        ToWin32ErrorCode := Win32ErrorCodes.ERROR_DS_DRA_INCONSISTENT_DIT;
    8444:
        ToWin32ErrorCode := Win32ErrorCodes.ERROR_DS_DRA_CONNECTION_FAILED;
    8445:
        ToWin32ErrorCode := Win32ErrorCodes.ERROR_DS_DRA_BAD_INSTANCE_TYPE;
    8446:
        ToWin32ErrorCode := Win32ErrorCodes.ERROR_DS_DRA_OUT_OF_MEM;
    8447:
        ToWin32ErrorCode := Win32ErrorCodes.ERROR_DS_DRA_MAIL_PROBLEM;
    8448:
        ToWin32ErrorCode := Win32ErrorCodes.ERROR_DS_DRA_REF_ALREADY_EXISTS;
    8449:
        ToWin32ErrorCode := Win32ErrorCodes.ERROR_DS_DRA_REF_NOT_FOUND;
    8450:
        ToWin32ErrorCode := Win32ErrorCodes.ERROR_DS_DRA_OBJ_IS_REP_SOURCE;
    8451:
        ToWin32ErrorCode := Win32ErrorCodes.ERROR_DS_DRA_DB_ERROR;
    8452:
        ToWin32ErrorCode := Win32ErrorCodes.ERROR_DS_DRA_NO_REPLICA;
    8453:
        ToWin32ErrorCode := Win32ErrorCodes.ERROR_DS_DRA_ACCESS_DENIED;
    8454:
        ToWin32ErrorCode := Win32ErrorCodes.ERROR_DS_DRA_NOT_SUPPORTED;
    8455:
        ToWin32ErrorCode := Win32ErrorCodes.ERROR_DS_DRA_RPC_CANCELLED;
    8456:
        ToWin32ErrorCode := Win32ErrorCodes.ERROR_DS_DRA_SOURCE_DISABLED;
    8457:
        ToWin32ErrorCode := Win32ErrorCodes.ERROR_DS_DRA_SINK_DISABLED;
    8458:
        ToWin32ErrorCode := Win32ErrorCodes.ERROR_DS_DRA_NAME_COLLISION;
    8459:
        ToWin32ErrorCode := Win32ErrorCodes.ERROR_DS_DRA_SOURCE_REINSTALLED;
    8460:
        ToWin32ErrorCode := Win32ErrorCodes.ERROR_DS_DRA_MISSING_PARENT;
    8461:
        ToWin32ErrorCode := Win32ErrorCodes.ERROR_DS_DRA_PREEMPTED;
    8462:
        ToWin32ErrorCode := Win32ErrorCodes.ERROR_DS_DRA_ABANDON_SYNC;
    8463:
        ToWin32ErrorCode := Win32ErrorCodes.ERROR_DS_DRA_SHUTDOWN;
    8464:
        ToWin32ErrorCode := Win32ErrorCodes.ERROR_DS_DRA_INCOMPATIBLE_PARTIAL_SET;
    8465:
        ToWin32ErrorCode := Win32ErrorCodes.ERROR_DS_DRA_SOURCE_IS_PARTIAL_REPLICA;
    8466:
        ToWin32ErrorCode := Win32ErrorCodes.ERROR_DS_DRA_EXTN_CONNECTION_FAILED;
    8467:
        ToWin32ErrorCode := Win32ErrorCodes.ERROR_DS_INSTALL_SCHEMA_MISMATCH;
    8468:
        ToWin32ErrorCode := Win32ErrorCodes.ERROR_DS_DUP_LINK_ID;
    8469:
        ToWin32ErrorCode := Win32ErrorCodes.ERROR_DS_NAME_ERROR_RESOLVING;
    8470:
        ToWin32ErrorCode := Win32ErrorCodes.ERROR_DS_NAME_ERROR_NOT_FOUND;
    8471:
        ToWin32ErrorCode := Win32ErrorCodes.ERROR_DS_NAME_ERROR_NOT_UNIQUE;
    8472:
        ToWin32ErrorCode := Win32ErrorCodes.ERROR_DS_NAME_ERROR_NO_MAPPING;
    8473:
        ToWin32ErrorCode := Win32ErrorCodes.ERROR_DS_NAME_ERROR_DOMAIN_ONLY;
    8474:
        ToWin32ErrorCode := Win32ErrorCodes.ERROR_DS_NAME_ERROR_NO_SYNTACTICAL_MAPPING;
    8475:
        ToWin32ErrorCode := Win32ErrorCodes.ERROR_DS_CONSTRUCTED_ATT_MOD;
    8476:
        ToWin32ErrorCode := Win32ErrorCodes.ERROR_DS_WRONG_OM_OBJ_CLASS;
    8477:
        ToWin32ErrorCode := Win32ErrorCodes.ERROR_DS_DRA_REPL_PENDING;
    8478:
        ToWin32ErrorCode := Win32ErrorCodes.ERROR_DS_DS_REQUIRED;
    8479:
        ToWin32ErrorCode := Win32ErrorCodes.ERROR_DS_INVALID_LDAP_DISPLAY_NAME;
    8480:
        ToWin32ErrorCode := Win32ErrorCodes.ERROR_DS_NON_BASE_SEARCH;
    8481:
        ToWin32ErrorCode := Win32ErrorCodes.ERROR_DS_CANT_RETRIEVE_ATTS;
    8482:
        ToWin32ErrorCode := Win32ErrorCodes.ERROR_DS_BACKLINK_WITHOUT_LINK;
    8483:
        ToWin32ErrorCode := Win32ErrorCodes.ERROR_DS_EPOCH_MISMATCH;
    8484:
        ToWin32ErrorCode := Win32ErrorCodes.ERROR_DS_SRC_NAME_MISMATCH;
    8485:
        ToWin32ErrorCode := Win32ErrorCodes.ERROR_DS_SRC_AND_DST_NC_IDENTICAL;
    8486:
        ToWin32ErrorCode := Win32ErrorCodes.ERROR_DS_DST_NC_MISMATCH;
    8487:
        ToWin32ErrorCode := Win32ErrorCodes.ERROR_DS_NOT_AUTHORITIVE_FOR_DST_NC;
    8488:
        ToWin32ErrorCode := Win32ErrorCodes.ERROR_DS_SRC_GUID_MISMATCH;
    8489:
        ToWin32ErrorCode := Win32ErrorCodes.ERROR_DS_CANT_MOVE_DELETED_OBJECT;
    8490:
        ToWin32ErrorCode := Win32ErrorCodes.ERROR_DS_PDC_OPERATION_IN_PROGRESS;
    8491:
        ToWin32ErrorCode := Win32ErrorCodes.ERROR_DS_CROSS_DOMAIN_CLEANUP_REQD;
    8492:
        ToWin32ErrorCode := Win32ErrorCodes.ERROR_DS_ILLEGAL_XDOM_MOVE_OPERATION;
    8493:
        ToWin32ErrorCode := Win32ErrorCodes.ERROR_DS_CANT_WITH_ACCT_GROUP_MEMBERSHPS;
    8494:
        ToWin32ErrorCode := Win32ErrorCodes.ERROR_DS_NC_MUST_HAVE_NC_PARENT;
    8495:
        ToWin32ErrorCode := Win32ErrorCodes.ERROR_DS_CR_IMPOSSIBLE_TO_VALIDATE;
    8496:
        ToWin32ErrorCode := Win32ErrorCodes.ERROR_DS_DST_DOMAIN_NOT_NATIVE;
    8497:
        ToWin32ErrorCode := Win32ErrorCodes.ERROR_DS_MISSING_INFRASTRUCTURE_CONTAINER;
    8498:
        ToWin32ErrorCode := Win32ErrorCodes.ERROR_DS_CANT_MOVE_ACCOUNT_GROUP;
    8499:
        ToWin32ErrorCode := Win32ErrorCodes.ERROR_DS_CANT_MOVE_RESOURCE_GROUP;
    8500:
        ToWin32ErrorCode := Win32ErrorCodes.ERROR_DS_INVALID_SEARCH_FLAG;
    8501:
        ToWin32ErrorCode := Win32ErrorCodes.ERROR_DS_NO_TREE_DELETE_ABOVE_NC;
    8502:
        ToWin32ErrorCode := Win32ErrorCodes.ERROR_DS_COULDNT_LOCK_TREE_FOR_DELETE;
    8503:
        ToWin32ErrorCode := Win32ErrorCodes.ERROR_DS_COULDNT_IDENTIFY_OBJECTS_FOR_TREE_DELETE;
    8504:
        ToWin32ErrorCode := Win32ErrorCodes.ERROR_DS_SAM_INIT_FAILURE;
    8505:
        ToWin32ErrorCode := Win32ErrorCodes.ERROR_DS_SENSITIVE_GROUP_VIOLATION;
    8506:
        ToWin32ErrorCode := Win32ErrorCodes.ERROR_DS_CANT_MOD_PRIMARYGROUPID;
    8507:
        ToWin32ErrorCode := Win32ErrorCodes.ERROR_DS_ILLEGAL_BASE_SCHEMA_MOD;
    8508:
        ToWin32ErrorCode := Win32ErrorCodes.ERROR_DS_NONSAFE_SCHEMA_CHANGE;
    8509:
        ToWin32ErrorCode := Win32ErrorCodes.ERROR_DS_SCHEMA_UPDATE_DISALLOWED;
    8510:
        ToWin32ErrorCode := Win32ErrorCodes.ERROR_DS_CANT_CREATE_UNDER_SCHEMA;
    8511:
        ToWin32ErrorCode := Win32ErrorCodes.ERROR_DS_INSTALL_NO_SRC_SCH_VERSION;
    8512:
        ToWin32ErrorCode := Win32ErrorCodes.ERROR_DS_INSTALL_NO_SCH_VERSION_IN_INIFILE;
    8513:
        ToWin32ErrorCode := Win32ErrorCodes.ERROR_DS_INVALID_GROUP_TYPE;
    8514:
        ToWin32ErrorCode := Win32ErrorCodes.ERROR_DS_NO_NEST_GLOBALGROUP_IN_MIXEDDOMAIN;
    8515:
        ToWin32ErrorCode := Win32ErrorCodes.ERROR_DS_NO_NEST_LOCALGROUP_IN_MIXEDDOMAIN;
    8516:
        ToWin32ErrorCode := Win32ErrorCodes.ERROR_DS_GLOBAL_CANT_HAVE_LOCAL_MEMBER;
    8517:
        ToWin32ErrorCode := Win32ErrorCodes.ERROR_DS_GLOBAL_CANT_HAVE_UNIVERSAL_MEMBER;
    8518:
        ToWin32ErrorCode := Win32ErrorCodes.ERROR_DS_UNIVERSAL_CANT_HAVE_LOCAL_MEMBER;
    8519:
        ToWin32ErrorCode := Win32ErrorCodes.ERROR_DS_GLOBAL_CANT_HAVE_CROSSDOMAIN_MEMBER;
    8520:
        ToWin32ErrorCode := Win32ErrorCodes.ERROR_DS_LOCAL_CANT_HAVE_CROSSDOMAIN_LOCAL_MEMBER;
    8521:
        ToWin32ErrorCode := Win32ErrorCodes.ERROR_DS_HAVE_PRIMARY_MEMBERS;
    8522:
        ToWin32ErrorCode := Win32ErrorCodes.ERROR_DS_STRING_SD_CONVERSION_FAILED;
    8523:
        ToWin32ErrorCode := Win32ErrorCodes.ERROR_DS_NAMING_MASTER_GC;
    8524:
        ToWin32ErrorCode := Win32ErrorCodes.ERROR_DS_LOOKUP_FAILURE;
    8525:
        ToWin32ErrorCode := Win32ErrorCodes.ERROR_DS_COULDNT_UPDATE_SPNS;
    8526:
        ToWin32ErrorCode := Win32ErrorCodes.ERROR_DS_CANT_RETRIEVE_SD;
    8527:
        ToWin32ErrorCode := Win32ErrorCodes.ERROR_DS_KEY_NOT_UNIQUE;
    8528:
        ToWin32ErrorCode := Win32ErrorCodes.ERROR_DS_WRONG_LINKED_ATT_SYNTAX;
    8529:
        ToWin32ErrorCode := Win32ErrorCodes.ERROR_DS_SAM_NEED_BOOTKEY_PASSWORD;
    8530:
        ToWin32ErrorCode := Win32ErrorCodes.ERROR_DS_SAM_NEED_BOOTKEY_FLOPPY;
    8531:
        ToWin32ErrorCode := Win32ErrorCodes.ERROR_DS_CANT_START;
    8532:
        ToWin32ErrorCode := Win32ErrorCodes.ERROR_DS_INIT_FAILURE;
    8533:
        ToWin32ErrorCode := Win32ErrorCodes.ERROR_DS_NO_PKT_PRIVACY_ON_CONNECTION;
    8534:
        ToWin32ErrorCode := Win32ErrorCodes.ERROR_DS_SOURCE_DOMAIN_IN_FOREST;
    8535:
        ToWin32ErrorCode := Win32ErrorCodes.ERROR_DS_DESTINATION_DOMAIN_NOT_IN_FOREST;
    8536:
        ToWin32ErrorCode := Win32ErrorCodes.ERROR_DS_DESTINATION_AUDITING_NOT_ENABLED;
    8537:
        ToWin32ErrorCode := Win32ErrorCodes.ERROR_DS_CANT_FIND_DC_FOR_SRC_DOMAIN;
    8538:
        ToWin32ErrorCode := Win32ErrorCodes.ERROR_DS_SRC_OBJ_NOT_GROUP_OR_USER;
    8539:
        ToWin32ErrorCode := Win32ErrorCodes.ERROR_DS_SRC_SID_EXISTS_IN_FOREST;
    8540:
        ToWin32ErrorCode := Win32ErrorCodes.ERROR_DS_SRC_AND_DST_OBJECT_CLASS_MISMATCH;
    8541:
        ToWin32ErrorCode := Win32ErrorCodes.ERROR_SAM_INIT_FAILURE;
    8542:
        ToWin32ErrorCode := Win32ErrorCodes.ERROR_DS_DRA_SCHEMA_INFO_SHIP;
    8543:
        ToWin32ErrorCode := Win32ErrorCodes.ERROR_DS_DRA_SCHEMA_CONFLICT;
    8544:
        ToWin32ErrorCode := Win32ErrorCodes.ERROR_DS_DRA_EARLIER_SCHEMA_CONLICT;
    8545:
        ToWin32ErrorCode := Win32ErrorCodes.ERROR_DS_DRA_OBJ_NC_MISMATCH;
    8546:
        ToWin32ErrorCode := Win32ErrorCodes.ERROR_DS_NC_STILL_HAS_DSAS;
    8547:
        ToWin32ErrorCode := Win32ErrorCodes.ERROR_DS_GC_REQUIRED;
    8548:
        ToWin32ErrorCode := Win32ErrorCodes.ERROR_DS_LOCAL_MEMBER_OF_LOCAL_ONLY;
    8549:
        ToWin32ErrorCode := Win32ErrorCodes.ERROR_DS_NO_FPO_IN_UNIVERSAL_GROUPS;
    8550:
        ToWin32ErrorCode := Win32ErrorCodes.ERROR_DS_CANT_ADD_TO_GC;
    8551:
        ToWin32ErrorCode := Win32ErrorCodes.ERROR_DS_NO_CHECKPOINT_WITH_PDC;
    8552:
        ToWin32ErrorCode := Win32ErrorCodes.ERROR_DS_SOURCE_AUDITING_NOT_ENABLED;
    8553:
        ToWin32ErrorCode := Win32ErrorCodes.ERROR_DS_CANT_CREATE_IN_NONDOMAIN_NC;
    8554:
        ToWin32ErrorCode := Win32ErrorCodes.ERROR_DS_INVALID_NAME_FOR_SPN;
    8555:
        ToWin32ErrorCode := Win32ErrorCodes.ERROR_DS_FILTER_USES_CONTRUCTED_ATTRS;
    8556:
        ToWin32ErrorCode := Win32ErrorCodes.ERROR_DS_UNICODEPWD_NOT_IN_QUOTES;
    8557:
        ToWin32ErrorCode := Win32ErrorCodes.ERROR_DS_MACHINE_ACCOUNT_QUOTA_EXCEEDED;
    8558:
        ToWin32ErrorCode := Win32ErrorCodes.ERROR_DS_MUST_BE_RUN_ON_DST_DC;
    8559:
        ToWin32ErrorCode := Win32ErrorCodes.ERROR_DS_SRC_DC_MUST_BE_SP4_OR_GREATER;
    8560:
        ToWin32ErrorCode := Win32ErrorCodes.ERROR_DS_CANT_TREE_DELETE_CRITICAL_OBJ;
    8561:
        ToWin32ErrorCode := Win32ErrorCodes.ERROR_DS_INIT_FAILURE_CONSOLE;
    8562:
        ToWin32ErrorCode := Win32ErrorCodes.ERROR_DS_SAM_INIT_FAILURE_CONSOLE;
    8563:
        ToWin32ErrorCode := Win32ErrorCodes.ERROR_DS_FOREST_VERSION_TOO_HIGH;
    8564:
        ToWin32ErrorCode := Win32ErrorCodes.ERROR_DS_DOMAIN_VERSION_TOO_HIGH;
    8565:
        ToWin32ErrorCode := Win32ErrorCodes.ERROR_DS_FOREST_VERSION_TOO_LOW;
    8566:
        ToWin32ErrorCode := Win32ErrorCodes.ERROR_DS_DOMAIN_VERSION_TOO_LOW;
    8567:
        ToWin32ErrorCode := Win32ErrorCodes.ERROR_DS_INCOMPATIBLE_VERSION;
    8568:
        ToWin32ErrorCode := Win32ErrorCodes.ERROR_DS_LOW_DSA_VERSION;
    8569:
        ToWin32ErrorCode := Win32ErrorCodes.ERROR_DS_NO_BEHAVIOR_VERSION_IN_MIXEDDOMAIN;
    8570:
        ToWin32ErrorCode := Win32ErrorCodes.ERROR_DS_NOT_SUPPORTED_SORT_ORDER;
    8571:
        ToWin32ErrorCode := Win32ErrorCodes.ERROR_DS_NAME_NOT_UNIQUE;
    8572:
        ToWin32ErrorCode := Win32ErrorCodes.ERROR_DS_MACHINE_ACCOUNT_CREATED_PRENT4;
    8573:
        ToWin32ErrorCode := Win32ErrorCodes.ERROR_DS_OUT_OF_VERSION_STORE;
    8574:
        ToWin32ErrorCode := Win32ErrorCodes.ERROR_DS_INCOMPATIBLE_CONTROLS_USED;
    8575:
        ToWin32ErrorCode := Win32ErrorCodes.ERROR_DS_NO_REF_DOMAIN;
    8576:
        ToWin32ErrorCode := Win32ErrorCodes.ERROR_DS_RESERVED_LINK_ID;
    8577:
        ToWin32ErrorCode := Win32ErrorCodes.ERROR_DS_LINK_ID_NOT_AVAILABLE;
    8578:
        ToWin32ErrorCode := Win32ErrorCodes.ERROR_DS_AG_CANT_HAVE_UNIVERSAL_MEMBER;
    8579:
        ToWin32ErrorCode := Win32ErrorCodes.ERROR_DS_MODIFYDN_DISALLOWED_BY_INSTANCE_TYPE;
    8580:
        ToWin32ErrorCode := Win32ErrorCodes.ERROR_DS_NO_OBJECT_MOVE_IN_SCHEMA_NC;
    8581:
        ToWin32ErrorCode := Win32ErrorCodes.ERROR_DS_MODIFYDN_DISALLOWED_BY_FLAG;
    8582:
        ToWin32ErrorCode := Win32ErrorCodes.ERROR_DS_MODIFYDN_WRONG_GRANDPARENT;
    8583:
        ToWin32ErrorCode := Win32ErrorCodes.ERROR_DS_NAME_ERROR_TRUST_REFERRAL;
    8584:
        ToWin32ErrorCode := Win32ErrorCodes.ERROR_NOT_SUPPORTED_ON_STANDARD_SERVER;
    8585:
        ToWin32ErrorCode := Win32ErrorCodes.ERROR_DS_CANT_ACCESS_REMOTE_PART_OF_AD;
    8586:
        ToWin32ErrorCode := Win32ErrorCodes.ERROR_DS_CR_IMPOSSIBLE_TO_VALIDATE_V2;
    8587:
        ToWin32ErrorCode := Win32ErrorCodes.ERROR_DS_THREAD_LIMIT_EXCEEDED;
    8588:
        ToWin32ErrorCode := Win32ErrorCodes.ERROR_DS_NOT_CLOSEST;
    9001:
        ToWin32ErrorCode := Win32ErrorCodes.DNS_ERROR_RCODE_FORMAT_ERROR;
    9002:
        ToWin32ErrorCode := Win32ErrorCodes.DNS_ERROR_RCODE_SERVER_FAILURE;
    9003:
        ToWin32ErrorCode := Win32ErrorCodes.DNS_ERROR_RCODE_NAME_ERROR;
    9004:
        ToWin32ErrorCode := Win32ErrorCodes.DNS_ERROR_RCODE_NOT_IMPLEMENTED;
    9005:
        ToWin32ErrorCode := Win32ErrorCodes.DNS_ERROR_RCODE_REFUSED;
    9006:
        ToWin32ErrorCode := Win32ErrorCodes.DNS_ERROR_RCODE_YXDOMAIN;
    9007:
        ToWin32ErrorCode := Win32ErrorCodes.DNS_ERROR_RCODE_YXRRSET;
    9008:
        ToWin32ErrorCode := Win32ErrorCodes.DNS_ERROR_RCODE_NXRRSET;
    9009:
        ToWin32ErrorCode := Win32ErrorCodes.DNS_ERROR_RCODE_NOTAUTH;
    9010:
        ToWin32ErrorCode := Win32ErrorCodes.DNS_ERROR_RCODE_NOTZONE;
    9016:
        ToWin32ErrorCode := Win32ErrorCodes.DNS_ERROR_RCODE_BADSIG;
    9017:
        ToWin32ErrorCode := Win32ErrorCodes.DNS_ERROR_RCODE_BADKEY;
    9018:
        ToWin32ErrorCode := Win32ErrorCodes.DNS_ERROR_RCODE_BADTIME;
    9501:
        ToWin32ErrorCode := Win32ErrorCodes.DNS_INFO_NO_RECORDS;
    9502:
        ToWin32ErrorCode := Win32ErrorCodes.DNS_ERROR_BAD_PACKET;
    9503:
        ToWin32ErrorCode := Win32ErrorCodes.DNS_ERROR_NO_PACKET;
    9504:
        ToWin32ErrorCode := Win32ErrorCodes.DNS_ERROR_RCODE;
    9505:
        ToWin32ErrorCode := Win32ErrorCodes.DNS_ERROR_UNSECURE_PACKET;
    9551:
        ToWin32ErrorCode := Win32ErrorCodes.DNS_ERROR_INVALID_TYPE;
    9552:
        ToWin32ErrorCode := Win32ErrorCodes.DNS_ERROR_INVALID_IP_ADDRESS;
    9553:
        ToWin32ErrorCode := Win32ErrorCodes.DNS_ERROR_INVALID_PROPERTY;
    9554:
        ToWin32ErrorCode := Win32ErrorCodes.DNS_ERROR_TRY_AGAIN_LATER;
    9555:
        ToWin32ErrorCode := Win32ErrorCodes.DNS_ERROR_NOT_UNIQUE;
    9556:
        ToWin32ErrorCode := Win32ErrorCodes.DNS_ERROR_NON_RFC_NAME;
    9557:
        ToWin32ErrorCode := Win32ErrorCodes.DNS_STATUS_FQDN;
    9558:
        ToWin32ErrorCode := Win32ErrorCodes.DNS_STATUS_DOTTED_NAME;
    9559:
        ToWin32ErrorCode := Win32ErrorCodes.DNS_STATUS_SINGLE_PART_NAME;
    9560:
        ToWin32ErrorCode := Win32ErrorCodes.DNS_ERROR_INVALID_NAME_CHAR;
    9561:
        ToWin32ErrorCode := Win32ErrorCodes.DNS_ERROR_NUMERIC_NAME;
    9601:
        ToWin32ErrorCode := Win32ErrorCodes.DNS_ERROR_ZONE_DOES_NOT_EXIST;
    9602:
        ToWin32ErrorCode := Win32ErrorCodes.DNS_ERROR_NO_ZONE_INFO;
    9603:
        ToWin32ErrorCode := Win32ErrorCodes.DNS_ERROR_INVALID_ZONE_OPERATION;
    9604:
        ToWin32ErrorCode := Win32ErrorCodes.DNS_ERROR_ZONE_CONFIGURATION_ERROR;
    9605:
        ToWin32ErrorCode := Win32ErrorCodes.DNS_ERROR_ZONE_HAS_NO_SOA_RECORD;
    9606:
        ToWin32ErrorCode := Win32ErrorCodes.DNS_ERROR_ZONE_HAS_NO_NS_RECORDS;
    9607:
        ToWin32ErrorCode := Win32ErrorCodes.DNS_ERROR_ZONE_LOCKED;
    9608:
        ToWin32ErrorCode := Win32ErrorCodes.DNS_ERROR_ZONE_CREATION_FAILED;
    9609:
        ToWin32ErrorCode := Win32ErrorCodes.DNS_ERROR_ZONE_ALREADY_EXISTS;
    9610:
        ToWin32ErrorCode := Win32ErrorCodes.DNS_ERROR_AUTOZONE_ALREADY_EXISTS;
    9611:
        ToWin32ErrorCode := Win32ErrorCodes.DNS_ERROR_INVALID_ZONE_TYPE;
    9612:
        ToWin32ErrorCode := Win32ErrorCodes.DNS_ERROR_SECONDARY_REQUIRES_MASTER_IP;
    9613:
        ToWin32ErrorCode := Win32ErrorCodes.DNS_ERROR_ZONE_NOT_SECONDARY;
    9614:
        ToWin32ErrorCode := Win32ErrorCodes.DNS_ERROR_NEED_SECONDARY_ADDRESSES;
    9615:
        ToWin32ErrorCode := Win32ErrorCodes.DNS_ERROR_WINS_INIT_FAILED;
    9616:
        ToWin32ErrorCode := Win32ErrorCodes.DNS_ERROR_NEED_WINS_SERVERS;
    9617:
        ToWin32ErrorCode := Win32ErrorCodes.DNS_ERROR_NBSTAT_INIT_FAILED;
    9618:
        ToWin32ErrorCode := Win32ErrorCodes.DNS_ERROR_SOA_DELETE_INVALID;
    9619:
        ToWin32ErrorCode := Win32ErrorCodes.DNS_ERROR_FORWARDER_ALREADY_EXISTS;
    9651:
        ToWin32ErrorCode := Win32ErrorCodes.DNS_ERROR_PRIMARY_REQUIRES_DATAFILE;
    9652:
        ToWin32ErrorCode := Win32ErrorCodes.DNS_ERROR_INVALID_DATAFILE_NAME;
    9653:
        ToWin32ErrorCode := Win32ErrorCodes.DNS_ERROR_DATAFILE_OPEN_FAILURE;
    9654:
        ToWin32ErrorCode := Win32ErrorCodes.DNS_ERROR_FILE_WRITEBACK_FAILED;
    9655:
        ToWin32ErrorCode := Win32ErrorCodes.DNS_ERROR_DATAFILE_PARSING;
    9701:
        ToWin32ErrorCode := Win32ErrorCodes.DNS_ERROR_RECORD_DOES_NOT_EXIST;
    9702:
        ToWin32ErrorCode := Win32ErrorCodes.DNS_ERROR_RECORD_FORMAT;
    9703:
        ToWin32ErrorCode := Win32ErrorCodes.DNS_ERROR_NODE_CREATION_FAILED;
    9704:
        ToWin32ErrorCode := Win32ErrorCodes.DNS_ERROR_UNKNOWN_RECORD_TYPE;
    9705:
        ToWin32ErrorCode := Win32ErrorCodes.DNS_ERROR_RECORD_TIMED_OUT;
    9706:
        ToWin32ErrorCode := Win32ErrorCodes.DNS_ERROR_NAME_NOT_IN_ZONE;
    9707:
        ToWin32ErrorCode := Win32ErrorCodes.DNS_ERROR_CNAME_LOOP;
    9708:
        ToWin32ErrorCode := Win32ErrorCodes.DNS_ERROR_NODE_IS_CNAME;
    9709:
        ToWin32ErrorCode := Win32ErrorCodes.DNS_ERROR_CNAME_COLLISION;
    9710:
        ToWin32ErrorCode := Win32ErrorCodes.DNS_ERROR_RECORD_ONLY_AT_ZONE_ROOT;
    9711:
        ToWin32ErrorCode := Win32ErrorCodes.DNS_ERROR_RECORD_ALREADY_EXISTS;
    9712:
        ToWin32ErrorCode := Win32ErrorCodes.DNS_ERROR_SECONDARY_DATA;
    9713:
        ToWin32ErrorCode := Win32ErrorCodes.DNS_ERROR_NO_CREATE_CACHE_DATA;
    9714:
        ToWin32ErrorCode := Win32ErrorCodes.DNS_ERROR_NAME_DOES_NOT_EXIST;
    9715:
        ToWin32ErrorCode := Win32ErrorCodes.DNS_WARNING_PTR_CREATE_FAILED;
    9716:
        ToWin32ErrorCode := Win32ErrorCodes.DNS_WARNING_DOMAIN_UNDELETED;
    9717:
        ToWin32ErrorCode := Win32ErrorCodes.DNS_ERROR_DS_UNAVAILABLE;
    9718:
        ToWin32ErrorCode := Win32ErrorCodes.DNS_ERROR_DS_ZONE_ALREADY_EXISTS;
    9719:
        ToWin32ErrorCode := Win32ErrorCodes.DNS_ERROR_NO_BOOTFILE_IF_DS_ZONE;
    9751:
        ToWin32ErrorCode := Win32ErrorCodes.DNS_INFO_AXFR_COMPLETE;
    9752:
        ToWin32ErrorCode := Win32ErrorCodes.DNS_ERROR_AXFR;
    9753:
        ToWin32ErrorCode := Win32ErrorCodes.DNS_INFO_ADDED_LOCAL_WINS;
    9801:
        ToWin32ErrorCode := Win32ErrorCodes.DNS_STATUS_CONTINUE_NEEDED;
    9851:
        ToWin32ErrorCode := Win32ErrorCodes.DNS_ERROR_NO_TCPIP;
    9852:
        ToWin32ErrorCode := Win32ErrorCodes.DNS_ERROR_NO_DNS_SERVERS;
    9901:
        ToWin32ErrorCode := Win32ErrorCodes.DNS_ERROR_DP_DOES_NOT_EXIST;
    9902:
        ToWin32ErrorCode := Win32ErrorCodes.DNS_ERROR_DP_ALREADY_EXISTS;
    9903:
        ToWin32ErrorCode := Win32ErrorCodes.DNS_ERROR_DP_NOT_ENLISTED;
    9904:
        ToWin32ErrorCode := Win32ErrorCodes.DNS_ERROR_DP_ALREADY_ENLISTED;
    10004:
        ToWin32ErrorCode := Win32ErrorCodes.WSAEINTR;
    10009:
        ToWin32ErrorCode := Win32ErrorCodes.WSAEBADF;
    10013:
        ToWin32ErrorCode := Win32ErrorCodes.WSAEACCES;
    10014:
        ToWin32ErrorCode := Win32ErrorCodes.WSAEFAULT;
    10022:
        ToWin32ErrorCode := Win32ErrorCodes.WSAEINVAL;
    10024:
        ToWin32ErrorCode := Win32ErrorCodes.WSAEMFILE;
    10035:
        ToWin32ErrorCode := Win32ErrorCodes.WSAEWOULDBLOCK;
    10036:
        ToWin32ErrorCode := Win32ErrorCodes.WSAEINPROGRESS;
    10037:
        ToWin32ErrorCode := Win32ErrorCodes.WSAEALREADY;
    10038:
        ToWin32ErrorCode := Win32ErrorCodes.WSAENOTSOCK;
    10039:
        ToWin32ErrorCode := Win32ErrorCodes.WSAEDESTADDRREQ;
    10040:
        ToWin32ErrorCode := Win32ErrorCodes.WSAEMSGSIZE;
    10041:
        ToWin32ErrorCode := Win32ErrorCodes.WSAEPROTOTYPE;
    10042:
        ToWin32ErrorCode := Win32ErrorCodes.WSAENOPROTOOPT;
    10043:
        ToWin32ErrorCode := Win32ErrorCodes.WSAEPROTONOSUPPORT;
    10044:
        ToWin32ErrorCode := Win32ErrorCodes.WSAESOCKTNOSUPPORT;
    10045:
        ToWin32ErrorCode := Win32ErrorCodes.WSAEOPNOTSUPP;
    10046:
        ToWin32ErrorCode := Win32ErrorCodes.WSAEPFNOSUPPORT;
    10047:
        ToWin32ErrorCode := Win32ErrorCodes.WSAEAFNOSUPPORT;
    10048:
        ToWin32ErrorCode := Win32ErrorCodes.WSAEADDRINUSE;
    10049:
        ToWin32ErrorCode := Win32ErrorCodes.WSAEADDRNOTAVAIL;
    10050:
        ToWin32ErrorCode := Win32ErrorCodes.WSAENETDOWN;
    10051:
        ToWin32ErrorCode := Win32ErrorCodes.WSAENETUNREACH;
    10052:
        ToWin32ErrorCode := Win32ErrorCodes.WSAENETRESET;
    10053:
        ToWin32ErrorCode := Win32ErrorCodes.WSAECONNABORTED;
    10054:
        ToWin32ErrorCode := Win32ErrorCodes.WSAECONNRESET;
    10055:
        ToWin32ErrorCode := Win32ErrorCodes.WSAENOBUFS;
    10056:
        ToWin32ErrorCode := Win32ErrorCodes.WSAEISCONN;
    10057:
        ToWin32ErrorCode := Win32ErrorCodes.WSAENOTCONN;
    10058:
        ToWin32ErrorCode := Win32ErrorCodes.WSAESHUTDOWN;
    10059:
        ToWin32ErrorCode := Win32ErrorCodes.WSAETOOMANYREFS;
    10060:
        ToWin32ErrorCode := Win32ErrorCodes.WSAETIMEDOUT;
    10061:
        ToWin32ErrorCode := Win32ErrorCodes.WSAECONNREFUSED;
    10062:
        ToWin32ErrorCode := Win32ErrorCodes.WSAELOOP;
    10063:
        ToWin32ErrorCode := Win32ErrorCodes.WSAENAMETOOLONG;
    10064:
        ToWin32ErrorCode := Win32ErrorCodes.WSAEHOSTDOWN;
    10065:
        ToWin32ErrorCode := Win32ErrorCodes.WSAEHOSTUNREACH;
    10066:
        ToWin32ErrorCode := Win32ErrorCodes.WSAENOTEMPTY;
    10067:
        ToWin32ErrorCode := Win32ErrorCodes.WSAEPROCLIM;
    10068:
        ToWin32ErrorCode := Win32ErrorCodes.WSAEUSERS;
    10069:
        ToWin32ErrorCode := Win32ErrorCodes.WSAEDQUOT;
    10070:
        ToWin32ErrorCode := Win32ErrorCodes.WSAESTALE;
    10071:
        ToWin32ErrorCode := Win32ErrorCodes.WSAEREMOTE;
    10091:
        ToWin32ErrorCode := Win32ErrorCodes.WSASYSNOTREADY;
    10092:
        ToWin32ErrorCode := Win32ErrorCodes.WSAVERNOTSUPPORTED;
    10093:
        ToWin32ErrorCode := Win32ErrorCodes.WSANOTINITIALISED;
    10101:
        ToWin32ErrorCode := Win32ErrorCodes.WSAEDISCON;
    10102:
        ToWin32ErrorCode := Win32ErrorCodes.WSAENOMORE;
    10103:
        ToWin32ErrorCode := Win32ErrorCodes.WSAECANCELLED;
    10104:
        ToWin32ErrorCode := Win32ErrorCodes.WSAEINVALIDPROCTABLE;
    10105:
        ToWin32ErrorCode := Win32ErrorCodes.WSAEINVALIDPROVIDER;
    10106:
        ToWin32ErrorCode := Win32ErrorCodes.WSAEPROVIDERFAILEDINIT;
    10107:
        ToWin32ErrorCode := Win32ErrorCodes.WSASYSCALLFAILURE;
    10108:
        ToWin32ErrorCode := Win32ErrorCodes.WSASERVICE_NOT_FOUND;
    10109:
        ToWin32ErrorCode := Win32ErrorCodes.WSATYPE_NOT_FOUND;
    10110:
        ToWin32ErrorCode := Win32ErrorCodes.WSA_E_NO_MORE;
    10111:
        ToWin32ErrorCode := Win32ErrorCodes.WSA_E_CANCELLED;
    10112:
        ToWin32ErrorCode := Win32ErrorCodes.WSAEREFUSED;
    11001:
        ToWin32ErrorCode := Win32ErrorCodes.WSAHOST_NOT_FOUND;
    11002:
        ToWin32ErrorCode := Win32ErrorCodes.WSATRY_AGAIN;
    11003:
        ToWin32ErrorCode := Win32ErrorCodes.WSANO_RECOVERY;
    11004:
        ToWin32ErrorCode := Win32ErrorCodes.WSANO_DATA;
    11005:
        ToWin32ErrorCode := Win32ErrorCodes.WSA_QOS_RECEIVERS;
    11006:
        ToWin32ErrorCode := Win32ErrorCodes.WSA_QOS_SENDERS;
    11007:
        ToWin32ErrorCode := Win32ErrorCodes.WSA_QOS_NO_SENDERS;
    11008:
        ToWin32ErrorCode := Win32ErrorCodes.WSA_QOS_NO_RECEIVERS;
    11009:
        ToWin32ErrorCode := Win32ErrorCodes.WSA_QOS_REQUEST_CONFIRMED;
    11010:
        ToWin32ErrorCode := Win32ErrorCodes.WSA_QOS_ADMISSION_FAILURE;
    11011:
        ToWin32ErrorCode := Win32ErrorCodes.WSA_QOS_POLICY_FAILURE;
    11012:
        ToWin32ErrorCode := Win32ErrorCodes.WSA_QOS_BAD_STYLE;
    11013:
        ToWin32ErrorCode := Win32ErrorCodes.WSA_QOS_BAD_OBJECT;
    11014:
        ToWin32ErrorCode := Win32ErrorCodes.WSA_QOS_TRAFFIC_CTRL_ERROR;
    11015:
        ToWin32ErrorCode := Win32ErrorCodes.WSA_QOS_GENERIC_ERROR;
    11016:
        ToWin32ErrorCode := Win32ErrorCodes.WSA_QOS_ESERVICETYPE;
    11017:
        ToWin32ErrorCode := Win32ErrorCodes.WSA_QOS_EFLOWSPEC;
    11018:
        ToWin32ErrorCode := Win32ErrorCodes.WSA_QOS_EPROVSPECBUF;
    11019:
        ToWin32ErrorCode := Win32ErrorCodes.WSA_QOS_EFILTERSTYLE;
    11020:
        ToWin32ErrorCode := Win32ErrorCodes.WSA_QOS_EFILTERTYPE;
    11021:
        ToWin32ErrorCode := Win32ErrorCodes.WSA_QOS_EFILTERCOUNT;
    11022:
        ToWin32ErrorCode := Win32ErrorCodes.WSA_QOS_EOBJLENGTH;
    11023:
        ToWin32ErrorCode := Win32ErrorCodes.WSA_QOS_EFLOWCOUNT;
    11024:
        ToWin32ErrorCode := Win32ErrorCodes.WSA_QOS_EUNKNOWNPSOBJ;
    11025:
        ToWin32ErrorCode := Win32ErrorCodes.WSA_QOS_EPOLICYOBJ;
    11026:
        ToWin32ErrorCode := Win32ErrorCodes.WSA_QOS_EFLOWDESC;
    11027:
        ToWin32ErrorCode := Win32ErrorCodes.WSA_QOS_EPSFLOWSPEC;
    11028:
        ToWin32ErrorCode := Win32ErrorCodes.WSA_QOS_EPSFILTERSPEC;
    11029:
        ToWin32ErrorCode := Win32ErrorCodes.WSA_QOS_ESDMODEOBJ;
    11030:
        ToWin32ErrorCode := Win32ErrorCodes.WSA_QOS_ESHAPERATEOBJ;
    11031:
        ToWin32ErrorCode := Win32ErrorCodes.WSA_QOS_RESERVED_PETYPE;
    12000:
        ToWin32ErrorCode := Win32ErrorCodes.ERROR_SXS_SECTION_NOT_FOUND;
    12001:
        ToWin32ErrorCode := Win32ErrorCodes.ERROR_SXS_CANT_GEN_ACTCTX;
    12002:
        ToWin32ErrorCode := Win32ErrorCodes.ERROR_SXS_INVALID_ACTCTXDATA_FORMAT;
    12003:
        ToWin32ErrorCode := Win32ErrorCodes.ERROR_SXS_ASSEMBLY_NOT_FOUND;
    12004:
        ToWin32ErrorCode := Win32ErrorCodes.ERROR_SXS_MANIFEST_FORMAT_ERROR;
    12005:
        ToWin32ErrorCode := Win32ErrorCodes.ERROR_SXS_MANIFEST_PARSE_ERROR;
    12006:
        ToWin32ErrorCode := Win32ErrorCodes.ERROR_SXS_ACTIVATION_CONTEXT_DISABLED;
    12007:
        ToWin32ErrorCode := Win32ErrorCodes.ERROR_SXS_KEY_NOT_FOUND;
    12008:
        ToWin32ErrorCode := Win32ErrorCodes.ERROR_SXS_VERSION_CONFLICT;
    12009:
        ToWin32ErrorCode := Win32ErrorCodes.ERROR_SXS_WRONG_SECTION_TYPE;
    12010:
        ToWin32ErrorCode := Win32ErrorCodes.ERROR_SXS_THREAD_QUERIES_DISABLED;
    12011:
        ToWin32ErrorCode := Win32ErrorCodes.ERROR_SXS_PROCESS_DEFAULT_ALREADY_SET;
    12012:
        ToWin32ErrorCode := Win32ErrorCodes.ERROR_SXS_UNKNOWN_ENCODING_GROUP;
    12013:
        ToWin32ErrorCode := Win32ErrorCodes.ERROR_SXS_UNKNOWN_ENCODING;
    12014:
        ToWin32ErrorCode := Win32ErrorCodes.ERROR_SXS_INVALID_XML_NAMESPACE_URI;
    12015:
        ToWin32ErrorCode := Win32ErrorCodes.ERROR_SXS_ROOT_MANIFEST_DEPENDENCY_NOT_INSTALLED;
    12016:
        ToWin32ErrorCode := Win32ErrorCodes.ERROR_SXS_LEAF_MANIFEST_DEPENDENCY_NOT_INSTALLED;
    12017:
        ToWin32ErrorCode := Win32ErrorCodes.ERROR_SXS_INVALID_ASSEMBLY_IDENTITY_ATTRIBUTE;
    12018:
        ToWin32ErrorCode := Win32ErrorCodes.ERROR_SXS_MANIFEST_MISSING_REQUIRED_DEFAULT_NAMESPACE;
    12019:
        ToWin32ErrorCode := Win32ErrorCodes.ERROR_SXS_MANIFEST_INVALID_REQUIRED_DEFAULT_NAMESPACE;
    12020:
        ToWin32ErrorCode :=
            Win32ErrorCodes.ERROR_SXS_PRIVATE_MANIFEST_CROSS_PATH_WITH_REPARSE_POINT;
    12021:
        ToWin32ErrorCode := Win32ErrorCodes.ERROR_SXS_DUPLICATE_DLL_NAME;
    12022:
        ToWin32ErrorCode := Win32ErrorCodes.ERROR_SXS_DUPLICATE_WINDOWCLASS_NAME;
    12023:
        ToWin32ErrorCode := Win32ErrorCodes.ERROR_SXS_DUPLICATE_CLSID;
    12024:
        ToWin32ErrorCode := Win32ErrorCodes.ERROR_SXS_DUPLICATE_IID;
    12025:
        ToWin32ErrorCode := Win32ErrorCodes.ERROR_SXS_DUPLICATE_TLBID;
    12026:
        ToWin32ErrorCode := Win32ErrorCodes.ERROR_SXS_DUPLICATE_PROGID;
    12027:
        ToWin32ErrorCode := Win32ErrorCodes.ERROR_SXS_DUPLICATE_ASSEMBLY_NAME;
    12028:
        ToWin32ErrorCode := Win32ErrorCodes.ERROR_SXS_FILE_HASH_MISMATCH;
    12029:
        ToWin32ErrorCode := Win32ErrorCodes.ERROR_SXS_POLICY_PARSE_ERROR;
    12030:
        ToWin32ErrorCode := Win32ErrorCodes.ERROR_SXS_XML_E_MISSINGQUOTE;
    12031:
        ToWin32ErrorCode := Win32ErrorCodes.ERROR_SXS_XML_E_COMMENTSYNTAX;
    12032:
        ToWin32ErrorCode := Win32ErrorCodes.ERROR_SXS_XML_E_BADSTARTNAMECHAR;
    12033:
        ToWin32ErrorCode := Win32ErrorCodes.ERROR_SXS_XML_E_BADNAMECHAR;
    12034:
        ToWin32ErrorCode := Win32ErrorCodes.ERROR_SXS_XML_E_BADCHARINSTRING;
    12035:
        ToWin32ErrorCode := Win32ErrorCodes.ERROR_SXS_XML_E_XMLDECLSYNTAX;
    12036:
        ToWin32ErrorCode := Win32ErrorCodes.ERROR_SXS_XML_E_BADCHARDATA;
    12037:
        ToWin32ErrorCode := Win32ErrorCodes.ERROR_SXS_XML_E_MISSINGWHITESPACE;
    12038:
        ToWin32ErrorCode := Win32ErrorCodes.ERROR_SXS_XML_E_EXPECTINGTAGEND;
    12039:
        ToWin32ErrorCode := Win32ErrorCodes.ERROR_SXS_XML_E_MISSINGSEMICOLON;
    12040:
        ToWin32ErrorCode := Win32ErrorCodes.ERROR_SXS_XML_E_UNBALANCEDPAREN;
    12041:
        ToWin32ErrorCode := Win32ErrorCodes.ERROR_SXS_XML_E_INTERNALERROR;
    12042:
        ToWin32ErrorCode := Win32ErrorCodes.ERROR_SXS_XML_E_UNEXPECTED_WHITESPACE;
    12043:
        ToWin32ErrorCode := Win32ErrorCodes.ERROR_SXS_XML_E_INCOMPLETE_ENCODING;
    12044:
        ToWin32ErrorCode := Win32ErrorCodes.ERROR_SXS_XML_E_MISSING_PAREN;
    12045:
        ToWin32ErrorCode := Win32ErrorCodes.ERROR_SXS_XML_E_EXPECTINGCLOSEQUOTE;
    12046:
        ToWin32ErrorCode := Win32ErrorCodes.ERROR_SXS_XML_E_MULTIPLE_COLONS;
    12047:
        ToWin32ErrorCode := Win32ErrorCodes.ERROR_SXS_XML_E_INVALID_DECIMAL;
    12048:
        ToWin32ErrorCode := Win32ErrorCodes.ERROR_SXS_XML_E_INVALID_HEXIDECIMAL;
    12049:
        ToWin32ErrorCode := Win32ErrorCodes.ERROR_SXS_XML_E_INVALID_UNICODE;
    12050:
        ToWin32ErrorCode := Win32ErrorCodes.ERROR_SXS_XML_E_WHITESPACEORQUESTIONMARK;
    12051:
        ToWin32ErrorCode := Win32ErrorCodes.ERROR_SXS_XML_E_UNEXPECTEDENDTAG;
    12052:
        ToWin32ErrorCode := Win32ErrorCodes.ERROR_SXS_XML_E_UNCLOSEDTAG;
    12053:
        ToWin32ErrorCode := Win32ErrorCodes.ERROR_SXS_XML_E_DUPLICATEATTRIBUTE;
    12054:
        ToWin32ErrorCode := Win32ErrorCodes.ERROR_SXS_XML_E_MULTIPLEROOTS;
    12055:
        ToWin32ErrorCode := Win32ErrorCodes.ERROR_SXS_XML_E_INVALIDATROOTLEVEL;
    12056:
        ToWin32ErrorCode := Win32ErrorCodes.ERROR_SXS_XML_E_BADXMLDECL;
    12057:
        ToWin32ErrorCode := Win32ErrorCodes.ERROR_SXS_XML_E_MISSINGROOT;
    12058:
        ToWin32ErrorCode := Win32ErrorCodes.ERROR_SXS_XML_E_UNEXPECTEDEOF;
    12059:
        ToWin32ErrorCode := Win32ErrorCodes.ERROR_SXS_XML_E_BADPEREFINSUBSET;
    12060:
        ToWin32ErrorCode := Win32ErrorCodes.ERROR_SXS_XML_E_UNCLOSEDSTARTTAG;
    12061:
        ToWin32ErrorCode := Win32ErrorCodes.ERROR_SXS_XML_E_UNCLOSEDENDTAG;
    12062:
        ToWin32ErrorCode := Win32ErrorCodes.ERROR_SXS_XML_E_UNCLOSEDSTRING;
    12063:
        ToWin32ErrorCode := Win32ErrorCodes.ERROR_SXS_XML_E_UNCLOSEDCOMMENT;
    12064:
        ToWin32ErrorCode := Win32ErrorCodes.ERROR_SXS_XML_E_UNCLOSEDDECL;
    12065:
        ToWin32ErrorCode := Win32ErrorCodes.ERROR_SXS_XML_E_UNCLOSEDCDATA;
    12066:
        ToWin32ErrorCode := Win32ErrorCodes.ERROR_SXS_XML_E_RESERVEDNAMESPACE;
    12067:
        ToWin32ErrorCode := Win32ErrorCodes.ERROR_SXS_XML_E_INVALIDENCODING;
    12068:
        ToWin32ErrorCode := Win32ErrorCodes.ERROR_SXS_XML_E_INVALIDSWITCH;
    12069:
        ToWin32ErrorCode := Win32ErrorCodes.ERROR_SXS_XML_E_BADXMLCASE;
    12070:
        ToWin32ErrorCode := Win32ErrorCodes.ERROR_SXS_XML_E_INVALID_STANDALONE;
    12071:
        ToWin32ErrorCode := Win32ErrorCodes.ERROR_SXS_XML_E_UNEXPECTED_STANDALONE;
    12072:
        ToWin32ErrorCode := Win32ErrorCodes.ERROR_SXS_XML_E_INVALID_VERSION;
    12073:
        ToWin32ErrorCode := Win32ErrorCodes.ERROR_SXS_XML_E_MISSINGEQUALS;
    13000:
        ToWin32ErrorCode := Win32ErrorCodes.ERROR_IPSEC_QM_POLICY_EXISTS;
    13001:
        ToWin32ErrorCode := Win32ErrorCodes.ERROR_IPSEC_QM_POLICY_NOT_FOUND;
    13002:
        ToWin32ErrorCode := Win32ErrorCodes.ERROR_IPSEC_QM_POLICY_IN_USE;
    13003:
        ToWin32ErrorCode := Win32ErrorCodes.ERROR_IPSEC_MM_POLICY_EXISTS;
    13004:
        ToWin32ErrorCode := Win32ErrorCodes.ERROR_IPSEC_MM_POLICY_NOT_FOUND;
    13005:
        ToWin32ErrorCode := Win32ErrorCodes.ERROR_IPSEC_MM_POLICY_IN_USE;
    13006:
        ToWin32ErrorCode := Win32ErrorCodes.ERROR_IPSEC_MM_FILTER_EXISTS;
    13007:
        ToWin32ErrorCode := Win32ErrorCodes.ERROR_IPSEC_MM_FILTER_NOT_FOUND;
    13008:
        ToWin32ErrorCode := Win32ErrorCodes.ERROR_IPSEC_TRANSPORT_FILTER_EXISTS;
    13009:
        ToWin32ErrorCode := Win32ErrorCodes.ERROR_IPSEC_TRANSPORT_FILTER_NOT_FOUND;
    13010:
        ToWin32ErrorCode := Win32ErrorCodes.ERROR_IPSEC_MM_AUTH_EXISTS;
    13011:
        ToWin32ErrorCode := Win32ErrorCodes.ERROR_IPSEC_MM_AUTH_NOT_FOUND;
    13012:
        ToWin32ErrorCode := Win32ErrorCodes.ERROR_IPSEC_MM_AUTH_IN_USE;
    13013:
        ToWin32ErrorCode := Win32ErrorCodes.ERROR_IPSEC_DEFAULT_MM_POLICY_NOT_FOUND;
    13014:
        ToWin32ErrorCode := Win32ErrorCodes.ERROR_IPSEC_DEFAULT_MM_AUTH_NOT_FOUND;
    13015:
        ToWin32ErrorCode := Win32ErrorCodes.ERROR_IPSEC_DEFAULT_QM_POLICY_NOT_FOUND;
    13016:
        ToWin32ErrorCode := Win32ErrorCodes.ERROR_IPSEC_TUNNEL_FILTER_EXISTS;
    13017:
        ToWin32ErrorCode := Win32ErrorCodes.ERROR_IPSEC_TUNNEL_FILTER_NOT_FOUND;
    13018:
        ToWin32ErrorCode := Win32ErrorCodes.ERROR_IPSEC_MM_FILTER_PENDING_DELETION;
    13019:
        ToWin32ErrorCode := Win32ErrorCodes.ERROR_IPSEC_TRANSPORT_FILTER_PENDING_DELETION;
    13020:
        ToWin32ErrorCode := Win32ErrorCodes.ERROR_IPSEC_TUNNEL_FILTER_PENDING_DELETION;
    13021:
        ToWin32ErrorCode := Win32ErrorCodes.ERROR_IPSEC_MM_POLICY_PENDING_DELETION;
    13022:
        ToWin32ErrorCode := Win32ErrorCodes.ERROR_IPSEC_MM_AUTH_PENDING_DELETION;
    13023:
        ToWin32ErrorCode := Win32ErrorCodes.ERROR_IPSEC_QM_POLICY_PENDING_DELETION;
    13801:
        ToWin32ErrorCode := Win32ErrorCodes.ERROR_IPSEC_IKE_AUTH_FAIL;
    13802:
        ToWin32ErrorCode := Win32ErrorCodes.ERROR_IPSEC_IKE_ATTRIB_FAIL;
    13803:
        ToWin32ErrorCode := Win32ErrorCodes.ERROR_IPSEC_IKE_NEGOTIATION_PENDING;
    13804:
        ToWin32ErrorCode := Win32ErrorCodes.ERROR_IPSEC_IKE_GENERAL_PROCESSING_ERROR;
    13805:
        ToWin32ErrorCode := Win32ErrorCodes.ERROR_IPSEC_IKE_TIMED_OUT;
    13806:
        ToWin32ErrorCode := Win32ErrorCodes.ERROR_IPSEC_IKE_NO_CERT;
    13807:
        ToWin32ErrorCode := Win32ErrorCodes.ERROR_IPSEC_IKE_SA_DELETED;
    13808:
        ToWin32ErrorCode := Win32ErrorCodes.ERROR_IPSEC_IKE_SA_REAPED;
    13809:
        ToWin32ErrorCode := Win32ErrorCodes.ERROR_IPSEC_IKE_MM_ACQUIRE_DROP;
    13810:
        ToWin32ErrorCode := Win32ErrorCodes.ERROR_IPSEC_IKE_QM_ACQUIRE_DROP;
    13811:
        ToWin32ErrorCode := Win32ErrorCodes.ERROR_IPSEC_IKE_QUEUE_DROP_MM;
    13812:
        ToWin32ErrorCode := Win32ErrorCodes.ERROR_IPSEC_IKE_QUEUE_DROP_NO_MM;
    13813:
        ToWin32ErrorCode := Win32ErrorCodes.ERROR_IPSEC_IKE_DROP_NO_RESPONSE;
    13814:
        ToWin32ErrorCode := Win32ErrorCodes.ERROR_IPSEC_IKE_MM_DELAY_DROP;
    13815:
        ToWin32ErrorCode := Win32ErrorCodes.ERROR_IPSEC_IKE_QM_DELAY_DROP;
    13816:
        ToWin32ErrorCode := Win32ErrorCodes.ERROR_IPSEC_IKE_ERROR;
    13817:
        ToWin32ErrorCode := Win32ErrorCodes.ERROR_IPSEC_IKE_CRL_FAILED;
    13818:
        ToWin32ErrorCode := Win32ErrorCodes.ERROR_IPSEC_IKE_INVALID_KEY_USAGE;
    13819:
        ToWin32ErrorCode := Win32ErrorCodes.ERROR_IPSEC_IKE_INVALID_CERT_TYPE;
    13820:
        ToWin32ErrorCode := Win32ErrorCodes.ERROR_IPSEC_IKE_NO_PRIVATE_KEY;
    13822:
        ToWin32ErrorCode := Win32ErrorCodes.ERROR_IPSEC_IKE_DH_FAIL;
    13824:
        ToWin32ErrorCode := Win32ErrorCodes.ERROR_IPSEC_IKE_INVALID_HEADER;
    13825:
        ToWin32ErrorCode := Win32ErrorCodes.ERROR_IPSEC_IKE_NO_POLICY;
    13826:
        ToWin32ErrorCode := Win32ErrorCodes.ERROR_IPSEC_IKE_INVALID_SIGNATURE;
    13827:
        ToWin32ErrorCode := Win32ErrorCodes.ERROR_IPSEC_IKE_KERBEROS_ERROR;
    13828:
        ToWin32ErrorCode := Win32ErrorCodes.ERROR_IPSEC_IKE_NO_PUBLIC_KEY;
    13829:
        ToWin32ErrorCode := Win32ErrorCodes.ERROR_IPSEC_IKE_PROCESS_ERR;
    13830:
        ToWin32ErrorCode := Win32ErrorCodes.ERROR_IPSEC_IKE_PROCESS_ERR_SA;
    13831:
        ToWin32ErrorCode := Win32ErrorCodes.ERROR_IPSEC_IKE_PROCESS_ERR_PROP;
    13832:
        ToWin32ErrorCode := Win32ErrorCodes.ERROR_IPSEC_IKE_PROCESS_ERR_TRANS;
    13833:
        ToWin32ErrorCode := Win32ErrorCodes.ERROR_IPSEC_IKE_PROCESS_ERR_KE;
    13834:
        ToWin32ErrorCode := Win32ErrorCodes.ERROR_IPSEC_IKE_PROCESS_ERR_ID;
    13835:
        ToWin32ErrorCode := Win32ErrorCodes.ERROR_IPSEC_IKE_PROCESS_ERR_CERT;
    13836:
        ToWin32ErrorCode := Win32ErrorCodes.ERROR_IPSEC_IKE_PROCESS_ERR_CERT_REQ;
    13837:
        ToWin32ErrorCode := Win32ErrorCodes.ERROR_IPSEC_IKE_PROCESS_ERR_HASH;
    13838:
        ToWin32ErrorCode := Win32ErrorCodes.ERROR_IPSEC_IKE_PROCESS_ERR_SIG;
    13839:
        ToWin32ErrorCode := Win32ErrorCodes.ERROR_IPSEC_IKE_PROCESS_ERR_NONCE;
    13840:
        ToWin32ErrorCode := Win32ErrorCodes.ERROR_IPSEC_IKE_PROCESS_ERR_NOTIFY;
    13841:
        ToWin32ErrorCode := Win32ErrorCodes.ERROR_IPSEC_IKE_PROCESS_ERR_DELETE;
    13842:
        ToWin32ErrorCode := Win32ErrorCodes.ERROR_IPSEC_IKE_PROCESS_ERR_VENDOR;
    13843:
        ToWin32ErrorCode := Win32ErrorCodes.ERROR_IPSEC_IKE_INVALID_PAYLOAD;
    13844:
        ToWin32ErrorCode := Win32ErrorCodes.ERROR_IPSEC_IKE_LOAD_SOFT_SA;
    13845:
        ToWin32ErrorCode := Win32ErrorCodes.ERROR_IPSEC_IKE_SOFT_SA_TORN_DOWN;
    13846:
        ToWin32ErrorCode := Win32ErrorCodes.ERROR_IPSEC_IKE_INVALID_COOKIE;
    13847:
        ToWin32ErrorCode := Win32ErrorCodes.ERROR_IPSEC_IKE_NO_PEER_CERT;
    13848:
        ToWin32ErrorCode := Win32ErrorCodes.ERROR_IPSEC_IKE_PEER_CRL_FAILED;
    13849:
        ToWin32ErrorCode := Win32ErrorCodes.ERROR_IPSEC_IKE_POLICY_CHANGE;
    13850:
        ToWin32ErrorCode := Win32ErrorCodes.ERROR_IPSEC_IKE_NO_MM_POLICY;
    13851:
        ToWin32ErrorCode := Win32ErrorCodes.ERROR_IPSEC_IKE_NOTCBPRIV;
    13852:
        ToWin32ErrorCode := Win32ErrorCodes.ERROR_IPSEC_IKE_SECLOADFAIL;
    13853:
        ToWin32ErrorCode := Win32ErrorCodes.ERROR_IPSEC_IKE_FAILSSPINIT;
    13854:
        ToWin32ErrorCode := Win32ErrorCodes.ERROR_IPSEC_IKE_FAILQUERYSSP;
    13855:
        ToWin32ErrorCode := Win32ErrorCodes.ERROR_IPSEC_IKE_SRVACQFAIL;
    13856:
        ToWin32ErrorCode := Win32ErrorCodes.ERROR_IPSEC_IKE_SRVQUERYCRED;
    13857:
        ToWin32ErrorCode := Win32ErrorCodes.ERROR_IPSEC_IKE_GETSPIFAIL;
    13858:
        ToWin32ErrorCode := Win32ErrorCodes.ERROR_IPSEC_IKE_INVALID_FILTER;
    13859:
        ToWin32ErrorCode := Win32ErrorCodes.ERROR_IPSEC_IKE_OUT_OF_MEMORY;
    13860:
        ToWin32ErrorCode := Win32ErrorCodes.ERROR_IPSEC_IKE_ADD_UPDATE_KEY_FAILED;
    13861:
        ToWin32ErrorCode := Win32ErrorCodes.ERROR_IPSEC_IKE_INVALID_POLICY;
    13862:
        ToWin32ErrorCode := Win32ErrorCodes.ERROR_IPSEC_IKE_UNKNOWN_DOI;
    13863:
        ToWin32ErrorCode := Win32ErrorCodes.ERROR_IPSEC_IKE_INVALID_SITUATION;
    13864:
        ToWin32ErrorCode := Win32ErrorCodes.ERROR_IPSEC_IKE_DH_FAILURE;
    13865:
        ToWin32ErrorCode := Win32ErrorCodes.ERROR_IPSEC_IKE_INVALID_GROUP;
    13866:
        ToWin32ErrorCode := Win32ErrorCodes.ERROR_IPSEC_IKE_ENCRYPT;
    13867:
        ToWin32ErrorCode := Win32ErrorCodes.ERROR_IPSEC_IKE_DECRYPT;
    13868:
        ToWin32ErrorCode := Win32ErrorCodes.ERROR_IPSEC_IKE_POLICY_MATCH;
    13869:
        ToWin32ErrorCode := Win32ErrorCodes.ERROR_IPSEC_IKE_UNSUPPORTED_ID;
    13870:
        ToWin32ErrorCode := Win32ErrorCodes.ERROR_IPSEC_IKE_INVALID_HASH;
    13871:
        ToWin32ErrorCode := Win32ErrorCodes.ERROR_IPSEC_IKE_INVALID_HASH_ALG;
    13872:
        ToWin32ErrorCode := Win32ErrorCodes.ERROR_IPSEC_IKE_INVALID_HASH_SIZE;
    13873:
        ToWin32ErrorCode := Win32ErrorCodes.ERROR_IPSEC_IKE_INVALID_ENCRYPT_ALG;
    13874:
        ToWin32ErrorCode := Win32ErrorCodes.ERROR_IPSEC_IKE_INVALID_AUTH_ALG;
    13875:
        ToWin32ErrorCode := Win32ErrorCodes.ERROR_IPSEC_IKE_INVALID_SIG;
    13876:
        ToWin32ErrorCode := Win32ErrorCodes.ERROR_IPSEC_IKE_LOAD_FAILED;
    13877:
        ToWin32ErrorCode := Win32ErrorCodes.ERROR_IPSEC_IKE_RPC_DELETE;
    13878:
        ToWin32ErrorCode := Win32ErrorCodes.ERROR_IPSEC_IKE_BENIGN_REINIT;
    13879:
        ToWin32ErrorCode := Win32ErrorCodes.ERROR_IPSEC_IKE_INVALID_RESPONDER_LIFETIME_NOTIFY;
    13880:
        ToWin32ErrorCode := Win32ErrorCodes.ERROR_IPSEC_IKE_QM_LIMIT_REAP;
    13881:
        ToWin32ErrorCode := Win32ErrorCodes.ERROR_IPSEC_IKE_INVALID_CERT_KEYLEN;
    13882:
        ToWin32ErrorCode := Win32ErrorCodes.ERROR_IPSEC_IKE_MM_LIMIT;
    13883:
        ToWin32ErrorCode := Win32ErrorCodes.ERROR_IPSEC_IKE_NEGOTIATION_DISABLED;
    13884:
        ToWin32ErrorCode := Win32ErrorCodes.ERROR_IPSEC_IKE_QM_LIMIT;
ELSE
    ToWin32ErrorCode := Win32ErrorCodes.ERR_UNKNOWN;
END_CASE

END_FUNCTION

(* stored: Version 1.1.0.1, ProductVersion 3.1.4024.11
   POU ToWin32ErrorCode: Id {fda7a771-6ab4-482e-ac10-0dfbc6445e30}, SpecialFunc None *)
